FUNCTION_BLOCK Test_TStreamAdd_Read_LREAL EXTENDS T_UnitTestBase
VAR
    Stream  : T_Stream(StreamLength := 2);
    ArgType : E_ArgTypeId := E_ArgTypeId.Type_LREAL;
END_VAR

{attribute 'analysis' := '-33'} // inhibit unused variable warning
METHOD RunTest
IF Retest THEN
    SUPER^.Init();
END_IF

IF TestCompleted THEN
    RETURN;
END_IF

F_Inc(CycleCount);
IF CycleCount > 1000 THEN
    Fail(Message := 'Timeout');
END_IF

Stream.Init(2);

// add a LREAL...
Stream.SetNextArgTypeId(ArgType);
Stream.Add_LREAL(1.234567891234);

Stream.SetReadPosition(0);

// check next arg type is correct...
AssertEquals_INT(Expected     := ArgType,
                           Actual       := Stream.GetNextArgTypeId(),
                           Message := 'Stream.GetNextArgTypeId()');

// check next value...	
AssertEquals_LREAL(Expected     := 1.234567891234,
                             Actual       := Stream.Read_LREAL(),
                             Delta        := 0.000000000001,
                             Message := 'Stream.Read_LREAL()');

// check we are at the end of the stream..							
AssertEquals_UDINT(Expected     := Stream.StreamLength,
                             Actual       := Stream.ReadPosition,
                             Message := 'Stream.ReadPosition');

TestCompleted := TRUE;
END_METHOD

END_FUNCTION_BLOCK

(* stored: Version 1.1.0.1, ProductVersion 3.1.4024.15
   POU Test_TStreamAdd_Read_LREAL: Id {75a7cde6-f38a-432c-a2b6-6088af846917}, SpecialFunc None
   Method RunTest: Id {1c79e0f8-8a8a-4a0f-b6ea-41acd73d44f1} *)
